FUNCTION_BLOCK FB_MatrixElementProduct_Test EXTENDS FB_TestSuite
VAR_INPUT
END_VAR
VAR_OUTPUT
END_VAR
VAR
END_VAR

WhenDifferentExpectError();
WhenmatchingExpectResult();

METHOD PRIVATE WhenDifferentExpectError
VAR_INPUT
END_VAR
VAR
	M1 : Matrix;
	M2 : Matrix;
	M3 : Matrix;
	Result : BOOL;
END_VAR
TEST('WhenDifferentExpectError');

// @TEST-RUN
M1.InitMagicSquare(3);
M2.InitMagicSquare(5);
Result := M3.AsElementProduct(M1,M2);

// @TEST-ASSERT
AssertFalse(Result,'Main function call was unexpectedly successful');

TEST_FINISHED();
END_METHOD

METHOD PRIVATE WhenMatchingExpectResult
VAR_INPUT
END_VAR
VAR
	M1 : Matrix;
	M2 : Matrix;
	M3 : Matrix;
	Result : BOOL;
END_VAR
TEST('WhenShrunkExpectDataRetained');

// @TEST-RUN
M1.InitMagicSquare(3);
M2.InitMagicSquare(3);
Result := M3.AsElementProduct(M1,M2);
M1.Power(2);

// @TEST-ASSERT
AssertTrue(Result,'Main function call was not successful');
AssertTrue(M3.IsEqual(M1),'Data was successfully multiplied');

TEST_FINISHED();
END_METHOD

END_FUNCTION_BLOCK

(* stored: Version 1.1.0.1, ProductVersion 3.1.4024.9
   POU FB_MatrixElementProduct_Test: Id {f04ce50a-919b-0b22-19c3-ecba2f551f8d}, SpecialFunc None
   Method WhenDifferentExpectError: Id {ab9d56c7-ba5b-00df-0667-a79c52cd33a2}
   Method WhenMatchingExpectResult: Id {64427d6c-abd8-0054-1ab6-597e00ab5274} *)
